{attribute 'no_explicit_call' := 'do not call this function block directly'} 
FUNCTION_BLOCK LoadFile EXTENDS ToolkitObject IMPLEMENTS IAction
VAR
	{attribute 'OPC.UA.DA' := '0'}
	_ClassName : STRING := __POUNAME();

	{attribute 'OPC.UA.DA' := '0'}
    _Load : Tc2_System.FB_FileLoad; 
	
	{attribute 'OPC.UA.DA' := '0'}
	_NeedStart : BOOL;
	{attribute 'OPC.UA.DA' := '0'}
	_Done : BOOL;
END_VAR

{attribute 'monitoring' := 'call'}
{attribute 'OPC.UA.DA.Property' := '1'}
{attribute 'OPC.UA.DA' := '1'}
PROPERTY AmsNetId : Tc2_System.T_AmsNetID
GET
AmsNetId := _Load.sNetId;
END_GET
SET
_Load.sNetId := AmsNetId;
END_SET
END_PROPERTY

{attribute 'monitoring' := 'call'}
{attribute 'OPC.UA.DA.Property' := '1'}
{attribute 'OPC.UA.DA.Access' := '1'}
PROPERTY Busy : BOOL
GET
Busy := _NeedStart OR_ELSE _Load.bBusy;
END_GET
END_PROPERTY

{attribute 'monitoring' := 'call'}
PROPERTY ClassName : STRING
GET
ClassName := _ClassName;
END_GET
END_PROPERTY

{attribute 'monitoring' := 'call'}
{attribute 'OPC.UA.DA.Property' := '1'}
{attribute 'OPC.UA.DA.Access' := '1'}
PROPERTY Done : BOOL
GET
Done := _Done;
END_GET
END_PROPERTY

{attribute 'monitoring' := 'call'}
{attribute 'OPC.UA.DA.Property' := '1'}
{attribute 'OPC.UA.DA.Access' := '1'}
PROPERTY Error : BOOL
GET
Error := _Load.bError;
END_GET
END_PROPERTY

METHOD Execute
VAR
	message : ERROR_MESSAGE;
END_VAR
IF _NeedStart OR_ELSE _Load.bBusy THEN
	_Load(bExecute := TRUE);
	_NeedStart := FALSE;
	
	IF _Load.bError THEN
		message := "An error occurred while loading the file '";
		WStringHelper.Append2(message, TO_WSTRING(_Load.sPathName), "'");	
		_LastException.Configure(message, __POUNAME(), ClassName, CurrentNamespace.Name, __POSITION(), _Load.nErrId).Throw();
	ELSIF NOT _Load.bBusy THEN
		_Done := TRUE;
	END_IF
END_IF
END_METHOD

{attribute 'monitoring' := 'call'}
{attribute 'OPC.UA.DA.Property' := '1'}
{attribute 'OPC.UA.DA.Access' := '1'}
PROPERTY LastException : REFERENCE TO Exception
GET
LastException REF= _LastException;
END_GET
END_PROPERTY

METHOD Start
VAR_INPUT
	filePath : Tc2_System.T_MaxString;
	targetBuffer : __System.AnyType;
END_VAR
_NeedStart := TRUE;
_Done := FALSE;
_Load.sPathName := filePath;
_Load.pReadBuff := targetBuffer.pValue;
_Load.cbReadLen := TO_UDINT(targetBuffer.diSize);

_LastException.Clear();
END_METHOD

{attribute 'monitoring' := 'call'}
{attribute 'OPC.UA.DA.Property' := '1'}
{attribute 'OPC.UA.DA' := '1'}
PROPERTY Timeout : TIME
GET
Timeout := _Load.tTimeout;
END_GET
SET
_Load.tTimeout := Timeout;
END_SET
END_PROPERTY

END_FUNCTION_BLOCK

(* stored: Version 1.1.0.1
   POU LoadFile: Id {9c614396-8297-440b-80fe-7fb36072951e}, SpecialFunc None
   Property AmsNetId: Id {20da3692-d6d8-4f78-82cf-66d6f738ff75}
   Get Get: Id {7e50120d-224a-4e29-ad24-b80fc65eb0f4}
   Set Set: Id {86ba0134-95b6-417c-8805-04bb775a2747}
   Property Busy: Id {b5d38962-4648-4e4e-bdf3-3e8ff480f904}
   Get Get: Id {4ca57017-31e7-4a62-9b35-18c53d3669fe}
   Property ClassName: Id {1bd161f1-6574-400f-82e8-23eb656b829c}
   Get Get: Id {06ad255f-09c3-4c01-ab4e-f78ad2e13312}
   Property Done: Id {8e88edbe-a6ac-4405-a322-5a96ecf18c11}
   Get Get: Id {d47f4c68-8919-45ba-8782-73f3ecca5af9}
   Property Error: Id {ec6a40f6-e867-4a0e-80d8-7fe28e0a4007}
   Get Get: Id {c40b661a-cfc1-4244-a8fe-60342b864a1c}
   Method Execute: Id {f951ef77-5cef-44e0-9ee2-db31a7da1635}
   Property LastException: Id {60cc9b60-61ac-4444-8c41-32730155c3b3}
   Get Get: Id {e216eb91-e570-403c-8d9a-8b608cc5abf4}
   Method Start: Id {1d918272-eb86-4106-9e83-1cd3bfe834f1}
   Property Timeout: Id {88df6ff3-eed5-4127-a5e9-cc3dae029abd}
   Get Get: Id {6d4f0f69-26a0-4a59-9a3a-4e25466c9423}
   Set Set: Id {da166a21-e0e0-4812-8c7f-5dcd9f1138f9} *)
